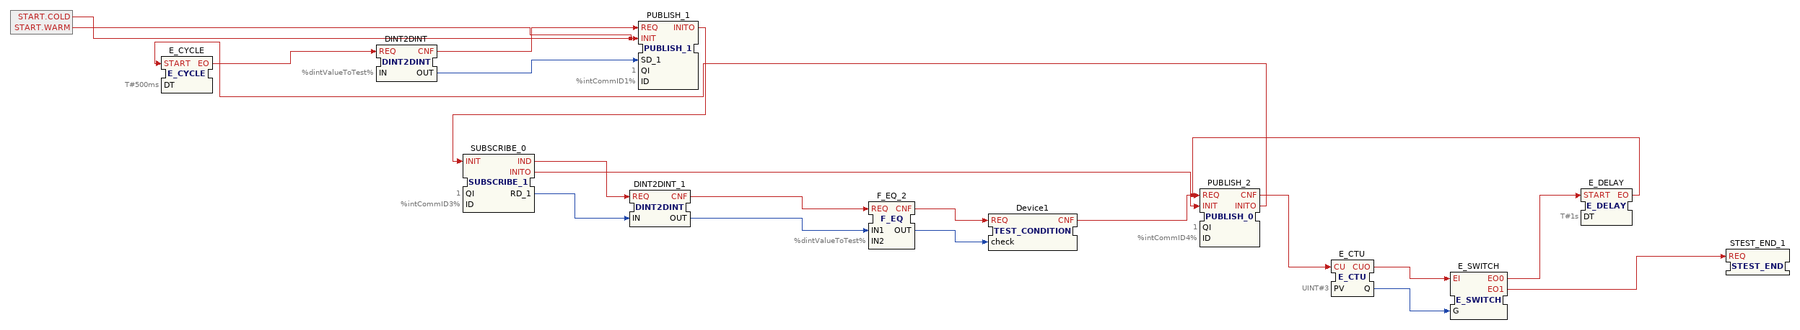
      FBS
        DINT2DINT : DINT2DINT(IN := %dintValueToTest%);
        E_CYCLE : E_CYCLE(DT := T#500ms);
        STEST_END_1 : STEST_END;
        PUBLISH_1 : PUBLISH_1(QI := 1, ID := %intCommID1%);
        F_EQ_2 : F_EQ(IN2 := %dintValueToTest%);
        Device1 : TEST_CONDITION;
        SUBSCRIBE_0 : SUBSCRIBE_1(QI := 1, ID := %intCommID3%);
        DINT2DINT_1 : DINT2DINT;
        E_DELAY : E_DELAY(DT := T#1s);
        PUBLISH_2 : PUBLISH_0(QI := 1, ID := %intCommID4%);
        E_CTU : E_CTU(PV := UINT#3);
        E_SWITCH : E_SWITCH;
      END_FBS
      EVENT_CONNECTIONS
        E_CYCLE.EO TO DINT2DINT.REQ;
        DINT2DINT.CNF TO PUBLISH_1.REQ;
        START.COLD TO PUBLISH_1.INIT;
        START.WARM TO PUBLISH_1.INIT;
        F_EQ_2.CNF TO Device1.REQ;
        PUBLISH_1.INITO TO SUBSCRIBE_0.INIT;
        SUBSCRIBE_0.IND TO DINT2DINT_1.REQ;
        DINT2DINT_1.CNF TO F_EQ_2.REQ;
        PUBLISH_2.CNF TO E_CTU.CU;
        E_CTU.CUO TO E_SWITCH.EI;
        E_SWITCH.EO0 TO E_DELAY.START;
        E_DELAY.EO TO PUBLISH_2.REQ;
        E_SWITCH.EO1 TO STEST_END_1.REQ;
        Device1.CNF TO PUBLISH_2.REQ;
        SUBSCRIBE_0.INITO TO PUBLISH_2.INIT;
        PUBLISH_2.INITO TO E_CYCLE.START;
      END_CONNECTIONS
      DATA_CONNECTIONS
        DINT2DINT.OUT TO PUBLISH_1.SD_1;
        F_EQ_2.OUT TO Device1.check;
        SUBSCRIBE_0.RD_1 TO DINT2DINT_1.IN;
        DINT2DINT_1.OUT TO F_EQ_2.IN1;
        E_CTU.Q TO E_SWITCH.G;
      END_CONNECTIONS
    END_RESOURCE
  END_DEVICE
  DEVICE Server : FORTE_PC(MGR_ID := "localhost:61501")
    {SET_ATTRIBUTE(Profile, HOLOBLOC)} (* device profile *)
    RESOURCE simpleServerTest : EMB_RES
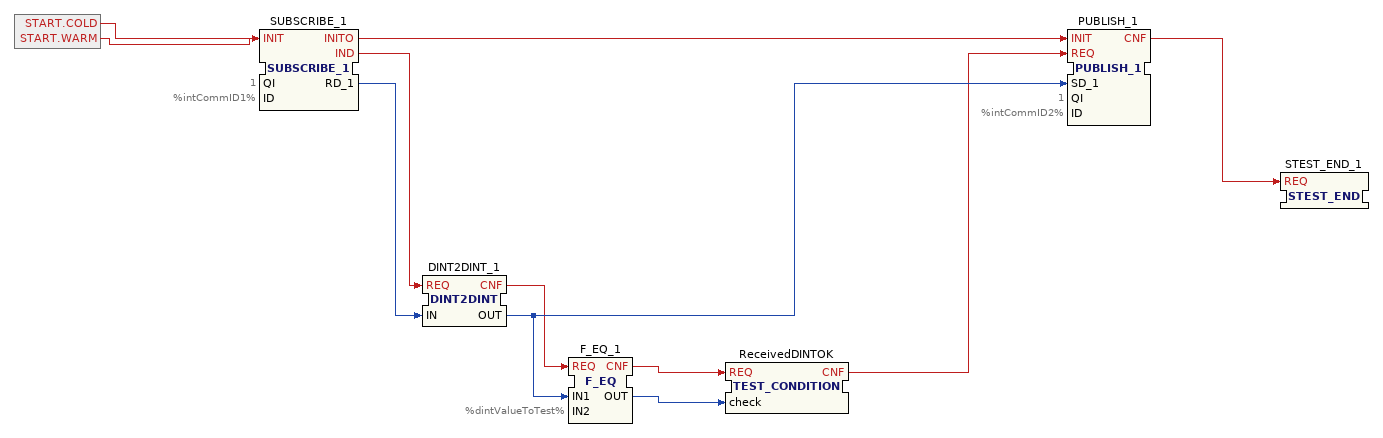
      FBS
        PUBLISH_1 : PUBLISH_1(QI := 1, ID := %intCommID2%);
        SUBSCRIBE_1 : SUBSCRIBE_1(QI := 1, ID := %intCommID1%);
        F_EQ_1 : F_EQ(IN2 := %dintValueToTest%);
        ReceivedDINTOK : TEST_CONDITION;
        DINT2DINT_1 : DINT2DINT;
        STEST_END_1 : STEST_END;
      END_FBS
      EVENT_CONNECTIONS
        START.COLD TO SUBSCRIBE_1.INIT;
        START.WARM TO SUBSCRIBE_1.INIT;
        SUBSCRIBE_1.INITO TO PUBLISH_1.INIT;
        F_EQ_1.CNF TO ReceivedDINTOK.REQ;
        DINT2DINT_1.CNF TO F_EQ_1.REQ;
        SUBSCRIBE_1.IND TO DINT2DINT_1.REQ;
        ReceivedDINTOK.CNF TO PUBLISH_1.REQ;
        PUBLISH_1.CNF TO STEST_END_1.REQ;
      END_CONNECTIONS
      DATA_CONNECTIONS
        F_EQ_1.OUT TO ReceivedDINTOK.check;
        DINT2DINT_1.OUT TO F_EQ_1.IN1;
        SUBSCRIBE_1.RD_1 TO DINT2DINT_1.IN;
        DINT2DINT_1.OUT TO PUBLISH_1.SD_1;
      END_CONNECTIONS
    END_RESOURCE
    RESOURCE multiDeviceEnd : EMB_RES
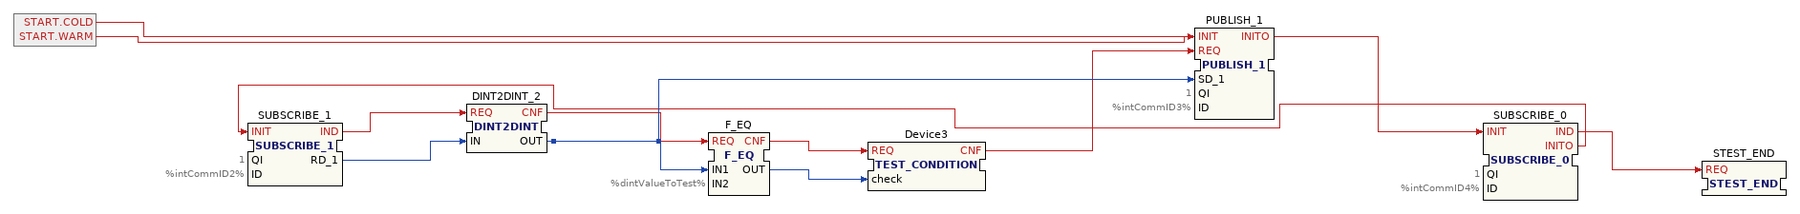
      FBS
        STEST_END : STEST_END;
        DINT2DINT_2 : DINT2DINT;
        F_EQ : F_EQ(IN2 := %dintValueToTest%);
        Device3 : TEST_CONDITION;
        SUBSCRIBE_1 : SUBSCRIBE_1(QI := 1, ID := %intCommID2%);
        SUBSCRIBE_0 : SUBSCRIBE_0(QI := 1, ID := %intCommID4%);
        PUBLISH_1 : PUBLISH_1(QI := 1, ID := %intCommID3%);
      END_FBS
      EVENT_CONNECTIONS
        DINT2DINT_2.CNF TO F_EQ.REQ;
        F_EQ.CNF TO Device3.REQ;
        SUBSCRIBE_1.IND TO DINT2DINT_2.REQ;
        SUBSCRIBE_0.IND TO STEST_END.REQ;
        SUBSCRIBE_0.INITO TO SUBSCRIBE_1.INIT;
        START.COLD TO PUBLISH_1.INIT;
        START.WARM TO PUBLISH_1.INIT;
        Device3.CNF TO PUBLISH_1.REQ;
        PUBLISH_1.INITO TO SUBSCRIBE_0.INIT;
      END_CONNECTIONS
      DATA_CONNECTIONS
        DINT2DINT_2.OUT TO F_EQ.IN1;
        F_EQ.OUT TO Device3.check;
        SUBSCRIBE_1.RD_1 TO DINT2DINT_2.IN;
        DINT2DINT_2.OUT TO PUBLISH_1.SD_1;
      END_CONNECTIONS
    END_RESOURCE
  END_DEVICE
  DEVICE CSVWriterTestDevice : FORTE_PC(MGR_ID := "localhost:61499")
    {SET_ATTRIBUTE(Profile, HOLOBLOC)} (* device profile *)
    RESOURCE normalExecution : EMB_RES
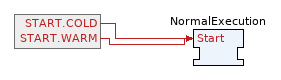
      SUBAPPLICATION NormalExecution
        EVENT_INPUT
          Start;
        END_EVENT
      END_SUBAPPLICATION
      EVENT_CONNECTIONS
        START.COLD TO NormalExecution.Start;
        START.WARM TO NormalExecution.Start;
      END_CONNECTIONS
    END_RESOURCE
    RESOURCE openAndNoClose : EMB_RES
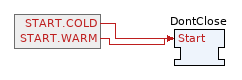
      SUBAPPLICATION DontClose
        EVENT_INPUT
          Start;
        END_EVENT
      END_SUBAPPLICATION
      EVENT_CONNECTIONS
        START.COLD TO DontClose.Start;
        START.WARM TO DontClose.Start;
      END_CONNECTIONS
    END_RESOURCE
    RESOURCE doubleInit : EMB_RES
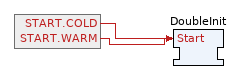
      SUBAPPLICATION DoubleInit
        EVENT_INPUT
          Start;
        END_EVENT
      END_SUBAPPLICATION
      EVENT_CONNECTIONS
        START.COLD TO DoubleInit.Start;
        START.WARM TO DoubleInit.Start;
      END_CONNECTIONS
    END_RESOURCE
    RESOURCE initDeinitNoWrite : EMB_RES
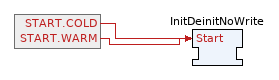
      SUBAPPLICATION InitDeinitNoWrite
        EVENT_INPUT
          Start;
        END_EVENT
      END_SUBAPPLICATION
      EVENT_CONNECTIONS
        START.COLD TO InitDeinitNoWrite.Start;
        START.WARM TO InitDeinitNoWrite.Start;
      END_CONNECTIONS
    END_RESOURCE
    RESOURCE closeNotOpened : EMB_RES
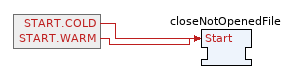
      SUBAPPLICATION closeNotOpenedFile
        EVENT_INPUT
          Start;
        END_EVENT
      END_SUBAPPLICATION
      EVENT_CONNECTIONS
        START.COLD TO closeNotOpenedFile.Start;
        START.WARM TO closeNotOpenedFile.Start;
      END_CONNECTIONS
    END_RESOURCE
    RESOURCE writeWithoutInit : EMB_RES
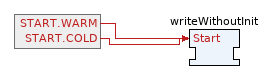
      SUBAPPLICATION writeWithoutInit
        EVENT_INPUT
          Start;
        END_EVENT
      END_SUBAPPLICATION
      EVENT_CONNECTIONS
        START.WARM TO writeWithoutInit.Start;
        START.COLD TO writeWithoutInit.Start;
      END_CONNECTIONS
    END_RESOURCE
    RESOURCE writeQIFalse : EMB_RES
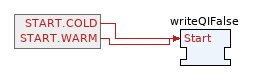
      SUBAPPLICATION writeQIFalse
        EVENT_INPUT
          Start;
        END_EVENT
      END_SUBAPPLICATION
      EVENT_CONNECTIONS
        START.COLD TO writeQIFalse.Start;
        START.WARM TO writeQIFalse.Start;
      END_CONNECTIONS
    END_RESOURCE
    RESOURCE normalExecutionMultiple : EMB_RES
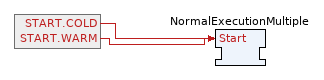
      SUBAPPLICATION NormalExecutionMultiple
        EVENT_INPUT
          Start;
        END_EVENT
      END_SUBAPPLICATION
      EVENT_CONNECTIONS
        START.COLD TO NormalExecutionMultiple.Start;
        START.WARM TO NormalExecutionMultiple.Start;
      END_CONNECTIONS
    END_RESOURCE
    RESOURCE noNameFile : EMB_RES
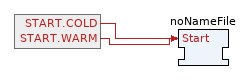
      SUBAPPLICATION noNameFile
        EVENT_INPUT
          Start;
        END_EVENT
      END_SUBAPPLICATION
      EVENT_CONNECTIONS
        START.COLD TO noNameFile.Start;
        START.WARM TO noNameFile.Start;
      END_CONNECTIONS
    END_RESOURCE
  END_DEVICE
  DEVICE MiddleSystem : FORTE_PC(MGR_ID := "localhost:61500")
    {SET_ATTRIBUTE(Profile, HOLOBLOC)} (* device profile *)
    RESOURCE multiDeviceMiddle : EMB_RES
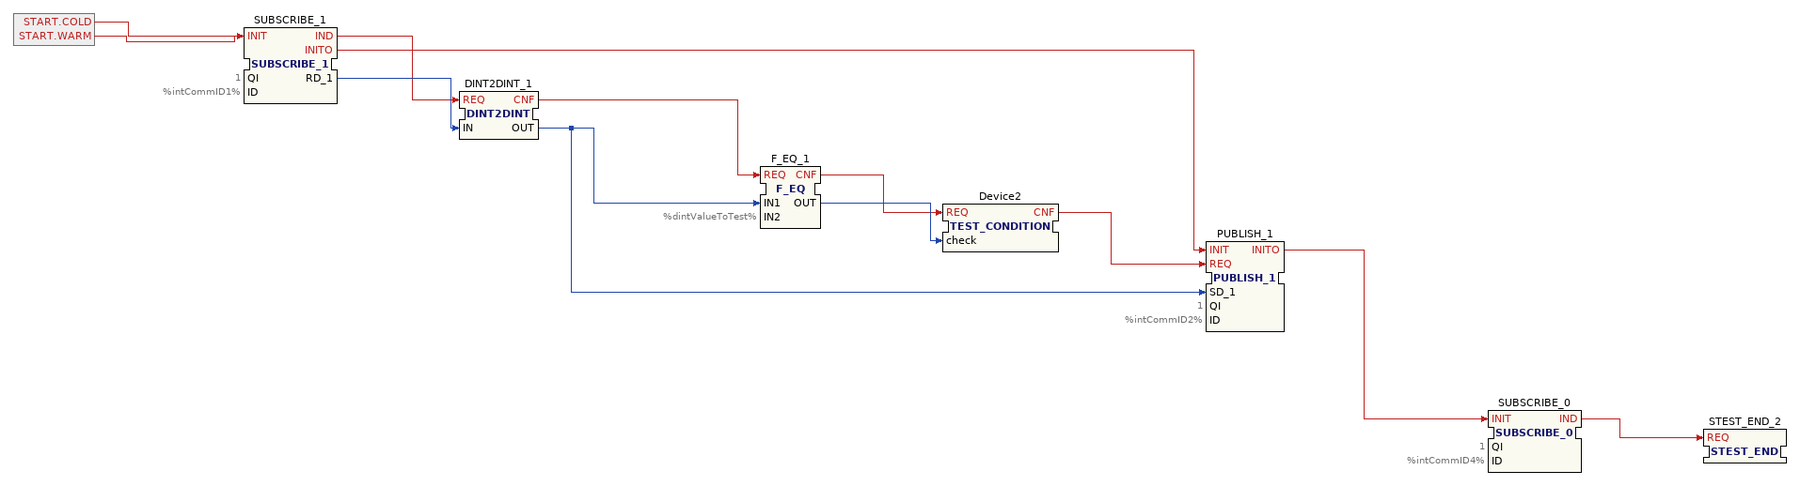
      FBS
        DINT2DINT_1 : DINT2DINT;
        F_EQ_1 : F_EQ(IN2 := %dintValueToTest%);
        Device2 : TEST_CONDITION;
        STEST_END_2 : STEST_END;
        SUBSCRIBE_1 : SUBSCRIBE_1(QI := 1, ID := %intCommID1%);
        PUBLISH_1 : PUBLISH_1(QI := 1, ID := %intCommID2%);
        SUBSCRIBE_0 : SUBSCRIBE_0(QI := 1, ID := %intCommID4%);
      END_FBS
      EVENT_CONNECTIONS
        F_EQ_1.CNF TO Device2.REQ;
        DINT2DINT_1.CNF TO F_EQ_1.REQ;
        SUBSCRIBE_1.IND TO DINT2DINT_1.REQ;
        START.COLD TO SUBSCRIBE_1.INIT;
        START.WARM TO SUBSCRIBE_1.INIT;
        SUBSCRIBE_1.INITO TO PUBLISH_1.INIT;
        Device2.CNF TO PUBLISH_1.REQ;
        SUBSCRIBE_0.IND TO STEST_END_2.REQ;
        PUBLISH_1.INITO TO SUBSCRIBE_0.INIT;
      END_CONNECTIONS
      DATA_CONNECTIONS
        DINT2DINT_1.OUT TO F_EQ_1.IN1;
        F_EQ_1.OUT TO Device2.check;
        SUBSCRIBE_1.RD_1 TO DINT2DINT_1.IN;
        DINT2DINT_1.OUT TO PUBLISH_1.SD_1;
      END_CONNECTIONS
    END_RESOURCE
  END_DEVICE
  MAPPINGS
    Timing.CSV_WRITER_1 ON DuT.TimingTestRes.CSV_WRITER_1;
    Timing.E_SR ON DuT.TimingTestRes.E_SR;
    Timing.E_SWITCH_2 ON DuT.TimingTestRes.E_SWITCH_2;
    Timing.Iterations ON DuT.TimingTestRes.Iterations;
    Timing.FBNuTest ON DuT.TimingTestRes.FBNuTest;
    Timing.STEST_END ON DuT.TimingTestRes.STEST_END;
    Timing.E_SWITCH ON DuT.TimingTestRes.E_SWITCH;
    Timing.E_StopWatch ON DuT.TimingTestRes.E_StopWatch;
    Soft_Pass_Example.NOT_ZERO ON DuT.Soft_Pass_Example.NOT_ZERO;
    Soft_Pass_Example.F_NOT ON DuT.Soft_Pass_Example.F_NOT;
    Soft_Pass_Example.BOOL2BOOL ON DuT.Soft_Pass_Example.BOOL2BOOL;
    Soft_Pass_Example.STEST_END_0_1 ON DuT.Soft_Pass_Example.STEST_END_0_1;
    Soft_Pass_Example.F_MUX_2 ON DuT.Soft_Pass_Example.F_MUX_2;
    Fail_Example.BOOL2BOOL_1_1_1 ON DuT.Fail_Example.BOOL2BOOL_1_1_1;
    Fail_Example.BOOL2BOOL_1 ON DuT.Fail_Example.BOOL2BOOL_1;
    Fail_Example.BOOL2BOOL_1_1 ON DuT.Fail_Example.BOOL2BOOL_1_1;
    Fail_Example.STEST_END_0 ON DuT.Fail_Example.STEST_END_0;
    Fail_Example.SHOULD_FAIL_1 ON DuT.Fail_Example.SHOULD_FAIL_1;
    Fail_Example.SHOULD_FAIL_2 ON DuT.Fail_Example.SHOULD_FAIL_2;
    Fail_Example.SHOULD_NOT_FAIL ON DuT.Fail_Example.SHOULD_NOT_FAIL;
    Hard_Pass_Example.STEST_END ON DuT.Hard_Pass_Example.STEST_END;
    Hard_Pass_Example.SHOULD_NOT_FAIL ON DuT.Hard_Pass_Example.SHOULD_NOT_FAIL;
    Hard_Pass_Example.BOOL2BOOL ON DuT.Hard_Pass_Example.BOOL2BOOL;
    DeInitCommFB.E_SR ON DuT.DeInitCommFB.E_SR;
    DeInitCommFB.E_SWITCH ON DuT.DeInitCommFB.E_SWITCH;
    DeInitCommFB.STEST_END ON DuT.DeInitCommFB.STEST_END;
    DeInitCommFB.PUBLISH_0 ON DuT.DeInitCommFB.PUBLISH_0;
    DeInitCommFB.E_SWITCH_1 ON DuT.DeInitCommFB.E_SWITCH_1;
    DeInitCommFB.E_SR_1 ON DuT.DeInitCommFB.E_SR_1;
    DeInitCommFB.E_SWITCH_2 ON DuT.DeInitCommFB.E_SWITCH_2;
    DeInitCommFB.E_SR_2 ON DuT.DeInitCommFB.E_SR_2;
    DeInitCommFB.E_SR_3 ON DuT.DeInitCommFB.E_SR_3;
    DeInitCommFB.E_SWITCH_3 ON DuT.DeInitCommFB.E_SWITCH_3;
    DeInitCommFB.PUBLISH_0_3 ON DuT.DeInitCommFB.PUBLISH_0_3;
    DeInitCommFB.PUBLISH_0_2 ON DuT.DeInitCommFB.PUBLISH_0_2;
    DeInitCommFB.PUBLISH_0_1 ON DuT.DeInitCommFB.PUBLISH_0_1;
    simpleCommunicationTest.WaitServer ON Client.simpleClientTest.WaitServer;
    simpleCommunicationTest.ReturnetValueOK ON Client.simpleClientTest.ReturnetValueOK;
    simpleCommunicationTest.F_EQ_1 ON Server.simpleServerTest.F_EQ_1;
    simpleCommunicationTest.F_EQ ON Client.simpleClientTest.F_EQ;
    simpleCommunicationTest.STEST_END ON Client.simpleClientTest.STEST_END;
    simpleCommunicationTest.DINT2DINT ON Client.simpleClientTest.DINT2DINT;
    simpleCommunicationTest.ReceivedDINTOK ON Server.simpleServerTest.ReceivedDINTOK;
    simpleCommunicationTest.DINT2DINT_1 ON Server.simpleServerTest.DINT2DINT_1;
    simpleCommunicationTest.DINT2DINT_2 ON Client.simpleClientTest.DINT2DINT_2;
    simpleCommunicationTest.STEST_END_1 ON Server.simpleServerTest.STEST_END_1;
    CSVWriterTests.NormalExecution ON CSVWriterTestDevice.normalExecution.NormalExecution;
    CSVWriterTests.DontClose ON CSVWriterTestDevice.openAndNoClose.DontClose;
    CSVWriterTests.DoubleInit ON CSVWriterTestDevice.doubleInit.DoubleInit;
    CSVWriterTests.InitDeinitNoWrite ON CSVWriterTestDevice.initDeinitNoWrite.InitDeinitNoWrite;
    CSVWriterTests.closeNotOpenedFile ON CSVWriterTestDevice.closeNotOpened.closeNotOpenedFile;
    CSVWriterTests.writeWithoutInit ON CSVWriterTestDevice.writeWithoutInit.writeWithoutInit;
    CSVWriterTests.writeQIFalse ON CSVWriterTestDevice.writeQIFalse.writeQIFalse;
    CSVWriterTests.NormalExecutionMultiple ON CSVWriterTestDevice.normalExecutionMultiple.NormalExecutionMultiple;
    CSVWriterTests.noNameFile ON CSVWriterTestDevice.noNameFile.noNameFile;
    MultiDevice.DINT2DINT ON Client.multiDeviceStart.DINT2DINT;
    MultiDevice.DINT2DINT_1 ON MiddleSystem.multiDeviceMiddle.DINT2DINT_1;
    MultiDevice.F_EQ_1 ON MiddleSystem.multiDeviceMiddle.F_EQ_1;
    MultiDevice.Device2 ON MiddleSystem.multiDeviceMiddle.Device2;
    MultiDevice.STEST_END ON Server.multiDeviceEnd.STEST_END;
    MultiDevice.DINT2DINT_2 ON Server.multiDeviceEnd.DINT2DINT_2;
    MultiDevice.F_EQ ON Server.multiDeviceEnd.F_EQ;
    MultiDevice.Device3 ON Server.multiDeviceEnd.Device3;
    MultiDevice.E_CYCLE ON Client.multiDeviceStart.E_CYCLE;
    MultiDevice.STEST_END_2 ON MiddleSystem.multiDeviceMiddle.STEST_END_2;
    MultiDevice.STEST_END_1 ON Client.multiDeviceStart.STEST_END_1;
    MultiDevice.F_EQ_2 ON Client.multiDeviceStart.F_EQ_2;
    MultiDevice.Device1 ON Client.multiDeviceStart.Device1;
  END_MAPPINGS
  SEGMENTS
    Ethernet : Ethernet;
  END_SEGMENTS
  LINKS
    Client => Ethernet;
    Server => Ethernet;
    MiddleSystem => Ethernet;
  END_LINKS
END_SYSTEM
